(* CODESYS project mobject-types.library
   Company: mobject
   DefaultNamespace: mobject-types
   Version: 0.1.0
   Placeholder: mobject-types
   Author: mobject dev team
   Title: mobject-types

Project tree, tasks and I/O mapping:
  libraries: mobject-collections, 1.1.0 (mobject); mobject-deserialization, 0.1.0 (mobject); mobject-disposable, 1.0.0 (mobject); mobject-enumerable, 1.1.0 (mobject); mobject-serialization, 0.4.0 (mobject); Tc2_System, * (Beckhoff Automation GmbH); Tc2_Utilities, * (Beckhoff Automation GmbH)
  _Internal/
    Datatype/
      function block AliasDatatypeBase [ST]: AddBaseType, BaseType, Identifier, IecType, SerializeTypeWith, SerializeWith, TryDeserializeFrom, TryResolveAsAliasType
      function block DatatypeBase [ST]: Accept, Address, ClearReference, Clone, IecType, SerializeTypeWith, SerializeWith, Size, TryCopy, TryDeserializeFrom, TryMakeReferenceTo, TryResolveAsAliasType, TryResolveAsStructuredType
      function block StructuredDatatypeBase [ST]: AddMember, Accept, GetMemberEnumerator, Identifier, IecType, SerializeTypeWith, SerializeWith, TryCopy, TryDeserializeFrom, TryGetMemberByName, TryResolveAsStructuredType
    DatatypeVisitor/
      interface I_DatatypeVisitor: VisitDatatype
    MembersHost/
      interface I_HostMembers: TryGetMemberByName
      function block MembersHost [ST]: Accept, AddMember, GetMemberEnumerator, SerializeTypeWith, SerializeWith, TryDeserializeFrom, TryGetMemberByName
  Datatype/
    Alias/
      function block _HRESULT [ST]: FB_init, SetBaseTypeReference, Address, ClearReference, Clone, Identifier, MakeReferenceTo, Size, TryMakeReferenceTo, Value
      function block _FLOAT [ST]: FB_init, SetBaseTypeReference, Address, ClearReference, Clone, Identifier, MakeReferenceTo, Size, TryMakeReferenceTo, Value
    Primitive/
      function block _BOOL [ST]: FB_init, Address, ClearReference, Clone, IecType, MakeReferenceTo, SerializeWith, Size, TryDeserializeFrom, TryMakeReferenceTo, Value
      function block _BYTE [ST]: FB_init, Address, ClearReference, Clone, IecType, MakeReferenceTo, SerializeWith, Size, TryDeserializeFrom, TryMakeReferenceTo, Value
      function block _DINT [ST]: FB_init, Address, ClearReference, Clone, IecType, MakeReferenceTo, SerializeWith, Size, TryDeserializeFrom, TryMakeReferenceTo, Value
      function block _DT [ST]: FB_init, Address, ClearReference, Clone, IecType, MakeReferenceTo, SerializeWith, Size, TryDeserializeFrom, TryMakeReferenceTo, Value
      function block _DWORD [ST]: FB_init, Address, ClearReference, Clone, IecType, MakeReferenceTo, SerializeWith, Size, TryDeserializeFrom, TryMakeReferenceTo, Value
      function block _INT [ST]: FB_init, Address, ClearReference, Clone, IecType, MakeReferenceTo, SerializeWith, Size, TryDeserializeFrom, TryMakeReferenceTo, Value
      function block _LINT [ST]: FB_init, Address, ClearReference, Clone, IecType, MakeReferenceTo, SerializeWith, Size, TryDeserializeFrom, TryMakeReferenceTo, Value
      function block _LREAL [ST]: FB_init, Address, ClearReference, Clone, IecType, MakeReferenceTo, SerializeWith, Size, TryDeserializeFrom, TryMakeReferenceTo, Value
      function block _LWORD [ST]: FB_init, Address, ClearReference, Clone, IecType, MakeReferenceTo, SerializeWith, Size, TryDeserializeFrom, TryMakeReferenceTo, Value
      function block _REAL [ST]: FB_init, Address, ClearReference, Clone, IecType, MakeReferenceTo, SerializeWith, Size, TryDeserializeFrom, TryMakeReferenceTo, Value
      function block _SINT [ST]: FB_init, Address, ClearReference, Clone, IecType, MakeReferenceTo, SerializeWith, Size, TryDeserializeFrom, TryMakeReferenceTo, Value
      function block _TIME_OF_DAY [ST]: FB_init, Address, ClearReference, Clone, IecType, MakeReferenceTo, SerializeWith, Size, TryDeserializeFrom, TryMakeReferenceTo, Value
      function block _TOD [ST]: FB_init, Address, ClearReference, Clone, IecType, MakeReferenceTo, SerializeWith, Size, TryDeserializeFrom, TryMakeReferenceTo, Value
      function block _UDINT [ST]: FB_init, Address, ClearReference, Clone, IecType, MakeReferenceTo, SerializeWith, Size, TryDeserializeFrom, TryMakeReferenceTo, Value
      function block _UINT [ST]: FB_init, Address, ClearReference, Clone, IecType, MakeReferenceTo, SerializeWith, Size, TryDeserializeFrom, TryMakeReferenceTo, Value
      function block _ULINT [ST]: FB_init, Address, ClearReference, Clone, IecType, MakeReferenceTo, SerializeWith, Size, TryDeserializeFrom, TryMakeReferenceTo, Value
      function block _USINT [ST]: FB_init, Address, ClearReference, Clone, IecType, MakeReferenceTo, SerializeWith, Size, TryDeserializeFrom, TryMakeReferenceTo, Value
      function block _WORD [ST]: FB_init, Address, ClearReference, Clone, IecType, MakeReferenceTo, SerializeWith, Size, TryDeserializeFrom, TryMakeReferenceTo, Value
    Structs/
      function block _TIMESTRUCT [ST]: FB_init, SetMemberReference, Address, ClearReference, Clone, Identifier, MakeReferenceTo, Size, TryMakeReferenceTo, Value, wDay, wDayOfWeek, wHour, wMilliseconds, wMinute, wMonth, wSecond, wYear
  DatatypePacks/
    function block PlcBasicDatatypePack [ST]: RegisterWith
  Datatypes/
    Base/
    function block Datatypes [ST]: SerializeAliasTypeWith, SerializePrimitiveTypeWith, SerializeStructuresTypeWith, GetAliasByIdentifier, GetPrimitiveByIecType, GetStructureByIdentifier, RegisterDatatype, SerializeTypeWith
  Interfaces/
    interface I_AliasDatatype: BaseType, Identifier
    interface I_Datatype: Accept, Address, ClearReference, Clone, IecType, SerializeTypeWith, Size, TryDeserializeFrom, TryMakeReferenceTo, TryResolveAsAliasType, TryResolveAsStructuredType
    interface I_DatatypePack: RegisterWith
    interface I_Datatypes: GetAliasByIdentifier, GetPrimitiveByIecType, GetStructureByIdentifier, RegisterDatatype, SerializeTypeWith
    interface I_StructuredDatatype: Identifier, TryGetMemberByName
*)

// _Internal/Datatype/AliasDatatypeBase
FUNCTION_BLOCK ABSTRACT AliasDatatypeBase EXTENDS DatatypeBase IMPLEMENTS I_AliasDatatype
VAR
	_baseType : I_Datatype;
END_VAR

METHOD PROTECTED AddBaseType
VAR_INPUT
	BaseType : I_Datatype;
END_VAR
_baseType := BaseType;
END_METHOD

PROPERTY PUBLIC BaseType : I_Datatype
GET
BaseType := _baseType;
END_GET
END_PROPERTY

PROPERTY PUBLIC ABSTRACT Identifier : T_MAXSTRING
GET
END_GET
END_PROPERTY

PROPERTY PUBLIC IecType : T_MAXSTRING
GET
IecType := 'ALIAS';
END_GET
END_PROPERTY

METHOD PUBLIC SerializeTypeWith
VAR_INPUT
	Serializer : I_Serializer;
END_VAR
Serializer.StartObject();
Serializer.AddKeyString('name',Identifier);
Serializer.AddKeyString('type',IecType);
Serializer.AddKey('baseType');
_baseType.SerializeTypeWith(Serializer);
Serializer.EndObject();
END_METHOD

METHOD PUBLIC SerializeWith
VAR_INPUT
	Serializer : I_Serializer;
END_VAR
_baseType.SerializeWith(Serializer);
END_METHOD

METHOD TryDeserializeFrom : BOOL
VAR_INPUT
	Deserializer : I_Deserializer;
	Feedback : I_DeserializerFeedback;
END_VAR
TryDeserializeFrom := _baseType.TryDeserializeFrom(Deserializer, Feedback);
END_METHOD

METHOD PUBLIC TryResolveAsAliasType : BOOL
VAR_INPUT
	Destination : REFERENCE TO I_AliasDatatype;
END_VAR
Destination := THIS^;
TryResolveAsAliasType := TRUE;
END_METHOD

END_FUNCTION_BLOCK

// _Internal/Datatype/DatatypeBase
{attribute 'linkalways'} 
{attribute 'no_explicit_call' := 'This FB is a CLASS and must be accessed using methods or properties'}
{attribute 'enable_dynamic_creation'}
FUNCTION_BLOCK ABSTRACT DatatypeBase EXTENDS Disposable IMPLEMENTS I_Datatype
VAR
END_VAR

METHOD PUBLIC Accept
VAR_INPUT
	Visitor : I_DatatypeVisitor;
END_VAR
Visitor.VisitDatatype(this^);
END_METHOD

PROPERTY PUBLIC ABSTRACT Address : PVOID
GET
END_GET
END_PROPERTY

METHOD PUBLIC ABSTRACT ClearReference
VAR_INPUT
END_VAR
END_METHOD

METHOD PUBLIC ABSTRACT Clone : I_Datatype
END_METHOD

PROPERTY PUBLIC ABSTRACT IecType : T_MAXSTRING
GET
END_GET
END_PROPERTY

METHOD PUBLIC SerializeTypeWith
VAR_INPUT
	Serializer : I_Serializer;
END_VAR
Serializer.StartObject();
Serializer.AddKeyString('type',IecType);
Serializer.EndObject();
END_METHOD

METHOD PUBLIC ABSTRACT SerializeWith
VAR_INPUT
	Serializer : I_Serializer;
END_VAR
END_METHOD

PROPERTY PUBLIC ABSTRACT Size : UDINT
GET
END_GET
END_PROPERTY

METHOD PUBLIC TryCopy : BOOL
VAR_INPUT
	Source : I_Datatype;
END_VAR
IF Source.IecType <> IecType THEN
	RETURN;
END_IF

memcpy(Address, Source.Address, Size);
END_METHOD

METHOD PUBLIC ABSTRACT TryDeserializeFrom : BOOL
VAR_INPUT
	Deserializer : I_Deserializer;
	Feedback : I_DeserializerFeedback;
END_VAR
END_METHOD

METHOD PUBLIC ABSTRACT TryMakeReferenceTo : BOOL
VAR_INPUT
	Target : I_Datatype;
END_VAR
END_METHOD

METHOD PUBLIC TryResolveAsAliasType : BOOL
VAR_INPUT
	Destination : REFERENCE TO I_AliasDatatype;
END_VAR
TryResolveAsAliasType := FALSE;
RETURN;
END_METHOD

METHOD PUBLIC TryResolveAsStructuredType : BOOL
VAR_INPUT
	Destination : REFERENCE TO I_StructuredDatatype;
END_VAR
TryResolveAsStructuredType := FALSE;
RETURN;
END_METHOD

END_FUNCTION_BLOCK

// Interfaces/I_Datatype
INTERFACE I_Datatype extends I_Serializable, I_Deserializable, I_Disposable

METHOD PUBLIC Accept
VAR_INPUT
	Visitor : I_DatatypeVisitor;
END_VAR
END_METHOD

PROPERTY PUBLIC Address : PVOID
GET
END_GET
END_PROPERTY

METHOD PUBLIC ClearReference
VAR_INPUT
END_VAR
END_METHOD

METHOD Clone : I_Datatype
END_METHOD

PROPERTY PUBLIC IecType : T_MAXSTRING
GET
END_GET
END_PROPERTY

METHOD PUBLIC SerializeTypeWith
VAR_INPUT
	Serializer : I_Serializer;
END_VAR
END_METHOD

PROPERTY PUBLIC Size : UDINT
GET
END_GET
END_PROPERTY

METHOD PUBLIC ABSTRACT TryDeserializeFrom : BOOL
VAR_INPUT
	Deserializer : I_Deserializer;
	Feedback : I_DeserializerFeedback;
END_VAR
END_METHOD

METHOD TryMakeReferenceTo : BOOL
VAR_INPUT
	Target : I_Datatype;
END_VAR
END_METHOD

METHOD PUBLIC TryResolveAsAliasType : BOOL
VAR_INPUT
	Destination : REFERENCE TO I_AliasDatatype;
END_VAR
END_METHOD

METHOD PUBLIC TryResolveAsStructuredType : BOOL
VAR_INPUT
	Destination : REFERENCE TO I_StructuredDatatype;
END_VAR
END_METHOD

END_INTERFACE

// _Internal/DatatypeVisitor/I_DatatypeVisitor
INTERFACE I_DatatypeVisitor

METHOD VisitDatatype
VAR_INPUT
	VisitingDatatype : I_Datatype;
END_VAR
END_METHOD

END_INTERFACE

// Interfaces/I_AliasDatatype
INTERFACE I_AliasDatatype EXTENDS I_Datatype

PROPERTY PUBLIC BaseType : I_Datatype
GET
END_GET
END_PROPERTY

PROPERTY PUBLIC Identifier : T_MAXSTRING
GET
END_GET
END_PROPERTY

END_INTERFACE

// Interfaces/I_StructuredDatatype
INTERFACE I_StructuredDatatype EXTENDS I_Datatype

PROPERTY PUBLIC Identifier : T_MAXSTRING
GET
END_GET
END_PROPERTY

METHOD PUBLIC TryGetMemberByName : BOOL
VAR_INPUT
	Name : T_MAXSTRING;
	Destination : REFERENCE TO I_Datatype;
END_VAR
END_METHOD

END_INTERFACE

// _Internal/Datatype/StructuredDatatypeBase
{attribute 'linkalways'} 
{attribute 'no_explicit_call' := 'This FB is a CLASS and must be accessed using methods or properties'}
{attribute 'enable_dynamic_creation'}
FUNCTION_BLOCK ABSTRACT StructuredDatatypeBase EXTENDS DatatypeBase IMPLEMENTS I_StructuredDatatype
VAR
	membersHost : MembersHost;
END_VAR

METHOD PROTECTED AddMember
VAR_INPUT
	MemberName : T_MAXSTRING;
	Member : I_Datatype;
END_VAR
membersHost.AddMember(MemberName, Member);
END_METHOD

METHOD PUBLIC Accept
VAR_INPUT
	Visitor : I_DatatypeVisitor;
END_VAR
Visitor.VisitDatatype(THIS^);
membersHost.Accept(Visitor);
END_METHOD

METHOD PUBLIC GetMemberEnumerator : I_KeyValueForwardEnumerator
VAR_INPUT
END_VAR
GetMemberEnumerator := membersHost.GetMemberEnumerator();
END_METHOD

PROPERTY PUBLIC ABSTRACT Identifier : T_MAXSTRING
GET
END_GET
END_PROPERTY

PROPERTY PUBLIC IecType : T_MAXSTRING
GET
IecType := 'STRUCT';
END_GET
END_PROPERTY

METHOD PUBLIC SerializeTypeWith
VAR_INPUT
	Serializer : I_Serializer;
END_VAR
Serializer.StartObject();
Serializer.AddKeyString('name',Identifier);
Serializer.AddKeyString('type',IecType);	
membersHost.SerializeTypeWith(Serializer);
Serializer.EndObject();
END_METHOD

METHOD PUBLIC SerializeWith
VAR_INPUT
	Serializer : I_Serializer;
END_VAR
Serializer.StartObject();
membersHost.SerializeWith(Serializer);
Serializer.EndObject();
END_METHOD

METHOD PUBLIC TryCopy : BOOL
VAR_INPUT
	Source : I_Datatype;
END_VAR
VAR
	SourceAsStructure : I_StructuredDatatype;
END_VAR
IF NOT Source.TryResolveAsStructuredType(SourceAsStructure) THEN
	RETURN;
END_IF

IF SourceAsStructure.Identifier <> Identifier THEN
	RETURN;
END_IF

memcpy(Address, Source.Address, Size);
END_METHOD

METHOD TryDeserializeFrom : BOOL
VAR_INPUT
	Deserializer : I_Deserializer;
	Feedback : I_DeserializerFeedback;
END_VAR
TryDeserializeFrom := membersHost.TryDeserializeFrom(Deserializer, Feedback);
END_METHOD

METHOD PUBLIC TryGetMemberByName : BOOL
VAR_INPUT
	Name : T_MAXSTRING;
	Destination : REFERENCE TO I_Datatype;
END_VAR
VAR
	member : I_Datatype;
END_VAR
IF NOT membersHost.TryGetMemberByName(Name, member) THEN 
	RETURN;
END_IF

Destination := member;
TryGetMemberByName := TRUE;
END_METHOD

METHOD PUBLIC TryResolveAsStructuredType : BOOL
VAR_INPUT
	Destination : REFERENCE TO I_StructuredDatatype;
END_VAR
Destination := THIS^;
TryResolveAsStructuredType := TRUE;
END_METHOD

END_FUNCTION_BLOCK

// _Internal/MembersHost/MembersHost
{attribute 'linkalways'} 
{attribute 'no_explicit_call' := 'This FB is a CLASS and must be accessed using methods or properties'}
{attribute 'enable_dynamic_creation'}
FUNCTION_BLOCK MembersHost IMPLEMENTS I_Serializable
VAR
	members : Dictionary;
END_VAR

METHOD PUBLIC Accept
VAR_INPUT
	Visitor : I_DatatypeVisitor;
END_VAR
VAR
	enumerator : I_ForwardEnumerator;
	member : I_Datatype;
END_VAR
enumerator := members.GetEnumerator();

WHILE (enumerator.MoveNext()) DO
	
	IF enumerator.TryGet(member) THEN
		member.Accept(Visitor);
	END_IF

END_WHILE

enumerator.Dispose();
END_METHOD

METHOD PUBLIC AddMember
VAR_INPUT
	MemberName : T_MAXSTRING;
	Member : I_Datatype;
END_VAR
members.AddOrUpdate(MemberName, Member);
END_METHOD

METHOD PUBLIC GetMemberEnumerator : I_KeyValueForwardEnumerator
VAR_INPUT
END_VAR
GetMemberEnumerator := members.GetKeyValueEnumerator();
END_METHOD

METHOD PUBLIC SerializeTypeWith
VAR_INPUT
	Serializer : I_Serializer;
END_VAR
VAR
	enumerator : I_KeyValueForwardEnumerator;
	member : I_Datatype;
END_VAR
IF members.Count = 0 THEN
	RETURN;
END_IF

Serializer.AddKey('members');
Serializer.StartObject();

enumerator := members.GetKeyValueEnumerator();

WHILE enumerator.MoveNext() DO
	IF enumerator.TryGet(member) THEN
		Serializer.AddKey(enumerator.Key);
		member.SerializeTypeWith(Serializer);
	END_IF
END_WHILE

enumerator.Dispose();

Serializer.EndObject();
END_METHOD

METHOD PUBLIC SerializeWith
VAR_INPUT
	Serializer : I_Serializer;
END_VAR
VAR
	enumerator : I_KeyValueForwardEnumerator;
	member : I_Datatype;
END_VAR
enumerator := members.GetKeyValueEnumerator();

WHILE enumerator.MoveNext() DO
	IF enumerator.TryGet(member) THEN
		Serializer.AddKey(enumerator.Key);
		member.SerializeWith(Serializer);
	END_IF
END_WHILE

enumerator.Dispose();
END_METHOD

METHOD PUBLIC TryDeserializeFrom : BOOL
VAR_INPUT
	Deserializer : I_Deserializer;
	Feedback : I_DeserializerFeedback;
END_VAR
VAR
	membersEnumerator : I_DeserializerObjectForwardEnumerator;
	member : I_Datatype;
END_VAR
membersEnumerator := Deserializer.GetObjectEnumerator();

WHILE membersEnumerator.MoveNext() DO
	
	IF NOT TryGetMemberByName(membersEnumerator.Key, member) THEN
		CONTINUE;
	END_IF
	
	IF NOT member.TryDeserializeFrom(membersEnumerator.Current, Feedback) THEN
		RETURN;
	END_IF

END_WHILE

membersEnumerator.Dispose();
TryDeserializeFrom := TRUE;
END_METHOD

METHOD PUBLIC TryGetMemberByName : BOOL
VAR_INPUT
	Name : T_MAXSTRING;
	Destination : REFERENCE TO I_Datatype;
END_VAR
VAR
	member : I_Datatype;
END_VAR
IF NOT members.TryGetValue(Name, member) THEN
	RETURN;
END_IF

Destination := member;
TryGetMemberByName := TRUE;
END_METHOD

END_FUNCTION_BLOCK

// _Internal/MembersHost/I_HostMembers
INTERFACE I_HostMembers EXTENDS __SYSTEM.IQueryInterface

METHOD PUBLIC TryGetMemberByName : BOOL
VAR_INPUT
	Name : T_MAXSTRING;
	Destination : REFERENCE TO I_Datatype;
END_VAR
END_METHOD

END_INTERFACE

// Datatype/Alias/_HRESULT
{attribute 'linkalways'} 
{attribute 'no_explicit_call' := 'This FB is a CLASS and must be accessed using methods or properties'}
{attribute 'enable_dynamic_creation'}
FUNCTION_BLOCK _HRESULT EXTENDS AliasDatatypeBase
VAR
	localData : HRESULT;
	activeData : REFERENCE TO HRESULT REF= localData;
	aliasBaseType : _DINT(localData);
END_VAR

METHOD FB_init : BOOL
VAR_INPUT
	bInitRetains : BOOL; // if TRUE, the retain variables are initialized (warm start / cold start)
	bInCopyCode : BOOL;  // if TRUE, the instance afterwards gets moved into the copy code (online change)
	InitialValue : HRESULT;
END_VAR
localData := InitialValue;
SetBaseTypeReference();
AddBaseType(aliasBaseType);
END_METHOD

METHOD PROTECTED SetBaseTypeReference
VAR_INPUT
END_VAR
aliasBaseType.MakeReferenceTo(activeData);
END_METHOD

PROPERTY PUBLIC Address : PVOID
GET
Address := ADR(activeData);
END_GET
END_PROPERTY

METHOD PUBLIC ClearReference
VAR_INPUT
END_VAR
activeData REF= localData;
SetBaseTypeReference();
END_METHOD

METHOD PUBLIC Clone : I_Datatype
VAR
    pClone : POINTER TO _HRESULT;
END_VAR
pClone := __NEW(_HRESULT(InitialValue := Value));
Clone := pClone^;
END_METHOD

PROPERTY PUBLIC Identifier : T_MAXSTRING
GET
Identifier := 'HRESULT';
END_GET
END_PROPERTY

METHOD PUBLIC MakeReferenceTo
VAR_INPUT
	ReferenceTarget : REFERENCE TO HRESULT;
END_VAR
activeData REF= ReferenceTarget;
SetBaseTypeReference();
END_METHOD

PROPERTY PUBLIC Size : UDINT
GET
Size := SIZEOF(activeData);
END_GET
END_PROPERTY

METHOD TryMakeReferenceTo : BOOL
VAR_INPUT
	Target : I_Datatype;
END_VAR
VAR
	pTargetData : POINTER TO HRESULT;
END_VAR
IF NOT (Target.IecType = IecType) THEN
	RETURN;
END_IF

pTargetData := Target.Address;
activeData REF= pTargetData^;
SetBaseTypeReference();
TryMakeReferenceTo := TRUE;
END_METHOD

PROPERTY PUBLIC Value : HRESULT
GET
Value := activeData;
END_GET
SET
activeData := Value;
END_SET
END_PROPERTY

END_FUNCTION_BLOCK

// Datatype/Primitive/_DINT
{attribute 'linkalways'} 
{attribute 'no_explicit_call' := 'This FB is a CLASS and must be accessed using methods or properties'}
{attribute 'enable_dynamic_creation'}
FUNCTION_BLOCK _DINT EXTENDS DatatypeBase
VAR
	localData : DINT;
	activeData : REFERENCE TO DINT REF= localData;
END_VAR

METHOD FB_init : BOOL
VAR_INPUT
	bInitRetains : BOOL; // if TRUE, the retain variables are initialized (warm start / cold start)
	bInCopyCode : BOOL;  // if TRUE, the instance afterwards gets moved into the copy code (online change)
	InitialValue : DINT;
END_VAR
localData := InitialValue;
END_METHOD

PROPERTY PUBLIC Address : PVOID
GET
Address := ADR(activeData);
END_GET
END_PROPERTY

METHOD PUBLIC ClearReference
VAR_INPUT
END_VAR
activeData REF= localData;
END_METHOD

METHOD PUBLIC Clone : I_Datatype
VAR
    pClone : POINTER TO _DINT;
END_VAR
pClone := __NEW(_DINT(InitialValue := Value));
Clone := pClone^;
END_METHOD

PROPERTY PUBLIC IecType : T_MAXSTRING
GET
IecType := 'DINT';
END_GET
END_PROPERTY

METHOD PUBLIC MakeReferenceTo
VAR_INPUT
	ReferenceTarget : REFERENCE TO DINT;
END_VAR
activeData REF= ReferenceTarget;
END_METHOD

METHOD PUBLIC SerializeWith
VAR_INPUT
	Serializer : I_Serializer;
END_VAR
Serializer.AddDint(activeData);
END_METHOD

PROPERTY PUBLIC Size : UDINT
GET
Size := SIZEOF(activeData);
END_GET
END_PROPERTY

METHOD TryDeserializeFrom : BOOL
VAR_INPUT
	Deserializer : I_Deserializer;
	Feedback : I_DeserializerFeedback;
END_VAR
TryDeserializeFrom := Deserializer.TryGetDint(activeData, Feedback);
END_METHOD

METHOD TryMakeReferenceTo : BOOL
VAR_INPUT
	Target : I_Datatype;
END_VAR
VAR
	pTargetData : POINTER TO DINT;
END_VAR
IF NOT (Target.IecType = IecType) THEN
	RETURN;
END_IF

pTargetData := Target.Address;
activeData REF= pTargetData^;
TryMakeReferenceTo := TRUE;
END_METHOD

PROPERTY PUBLIC Value : DINT
GET
Value := activeData;
END_GET
SET
activeData := Value;
END_SET
END_PROPERTY

END_FUNCTION_BLOCK

// Datatype/Alias/_FLOAT
{attribute 'linkalways'} 
{attribute 'no_explicit_call' := 'This FB is a CLASS and must be accessed using methods or properties'}
{attribute 'enable_dynamic_creation'}
FUNCTION_BLOCK _FLOAT EXTENDS AliasDatatypeBase
VAR
	localData : FLOAT;
	activeData : REFERENCE TO FLOAT REF= localData;
	aliasBaseType : _LREAL(localData);
END_VAR

METHOD FB_init : BOOL
VAR_INPUT
	bInitRetains : BOOL; // if TRUE, the retain variables are initialized (warm start / cold start)
	bInCopyCode : BOOL;  // if TRUE, the instance afterwards gets moved into the copy code (online change)
	InitialValue : FLOAT;
END_VAR
localData := InitialValue;
SetBaseTypeReference();
AddBaseType(aliasBaseType);
END_METHOD

METHOD PROTECTED SetBaseTypeReference
VAR_INPUT
END_VAR
aliasBaseType.MakeReferenceTo(activeData);
END_METHOD

PROPERTY PUBLIC Address : PVOID
GET
Address := ADR(activeData);
END_GET
END_PROPERTY

METHOD PUBLIC ClearReference
VAR_INPUT
END_VAR
activeData REF= localData;
SetBaseTypeReference();
END_METHOD

METHOD PUBLIC Clone : I_Datatype
VAR
    pClone : POINTER TO _FLOAT;
END_VAR
pClone := __NEW(_FLOAT(InitialValue := Value));
Clone := pClone^;
END_METHOD

PROPERTY PUBLIC Identifier : T_MAXSTRING
GET
Identifier := 'FLOAT';
END_GET
END_PROPERTY

METHOD PUBLIC MakeReferenceTo
VAR_INPUT
	ReferenceTarget : REFERENCE TO FLOAT;
END_VAR
activeData REF= ReferenceTarget;
SetBaseTypeReference();
END_METHOD

PROPERTY PUBLIC Size : UDINT
GET
Size := SIZEOF(activeData);
END_GET
END_PROPERTY

METHOD TryMakeReferenceTo : BOOL
VAR_INPUT
	Target : I_Datatype;
END_VAR
VAR
	pTargetData : POINTER TO FLOAT;
END_VAR
IF NOT (Target.IecType = IecType) THEN
	RETURN;
END_IF

pTargetData := Target.Address;
activeData REF= pTargetData^;
SetBaseTypeReference();
TryMakeReferenceTo := TRUE;
END_METHOD

PROPERTY PUBLIC Value : FLOAT
GET
Value := activeData;
END_GET
SET
activeData := Value;
END_SET
END_PROPERTY

END_FUNCTION_BLOCK

// Datatype/Primitive/_LREAL
{attribute 'linkalways'} 
{attribute 'no_explicit_call' := 'This FB is a CLASS and must be accessed using methods or properties'}
{attribute 'enable_dynamic_creation'}
FUNCTION_BLOCK _LREAL EXTENDS DatatypeBase
VAR
	localData : LREAL;
	activeData : REFERENCE TO LREAL REF= localData;
END_VAR

METHOD FB_init : BOOL
VAR_INPUT
	bInitRetains : BOOL; // if TRUE, the retain variables are initialized (warm start / cold start)
	bInCopyCode : BOOL;  // if TRUE, the instance afterwards gets moved into the copy code (online change)
	InitialValue : LREAL;
END_VAR
localData := InitialValue;
END_METHOD

PROPERTY PUBLIC Address : PVOID
GET
Address := ADR(activeData);
END_GET
END_PROPERTY

METHOD PUBLIC ClearReference
VAR_INPUT
END_VAR
activeData REF= localData;
END_METHOD

METHOD PUBLIC Clone : I_Datatype
VAR
    pClone : POINTER TO _LREAL;
END_VAR
pClone := __NEW(_LREAL(InitialValue := Value));
Clone := pClone^;
END_METHOD

PROPERTY PUBLIC IecType : T_MAXSTRING
GET
IecType := 'LREAL';
END_GET
END_PROPERTY

METHOD PUBLIC MakeReferenceTo
VAR_INPUT
	ReferenceTarget : REFERENCE TO LREAL;
END_VAR
activeData REF= ReferenceTarget;
END_METHOD

METHOD PUBLIC SerializeWith
VAR_INPUT
	Serializer : I_Serializer;
END_VAR
Serializer.AddLreal(activeData);
END_METHOD

PROPERTY PUBLIC Size : UDINT
GET
Size := SIZEOF(activeData);
END_GET
END_PROPERTY

METHOD TryDeserializeFrom : BOOL
VAR_INPUT
	Deserializer : I_Deserializer;
	Feedback : I_DeserializerFeedback;
END_VAR
TryDeserializeFrom := Deserializer.TryGetLreal(activeData, Feedback);
END_METHOD

METHOD TryMakeReferenceTo : BOOL
VAR_INPUT
	Target : I_Datatype;
END_VAR
VAR
	pTargetData : POINTER TO LREAL;
END_VAR
IF NOT (Target.IecType = IecType) THEN
	RETURN;
END_IF

pTargetData := Target.Address;
activeData REF= pTargetData^;
TryMakeReferenceTo := TRUE;
END_METHOD

PROPERTY PUBLIC Value : LREAL
GET
Value := activeData;
END_GET
SET
activeData := Value;
END_SET
END_PROPERTY

END_FUNCTION_BLOCK

// Datatype/Primitive/_BOOL
{attribute 'linkalways'} 
{attribute 'no_explicit_call' := 'This FB is a CLASS and must be accessed using methods or properties'}
{attribute 'enable_dynamic_creation'}
FUNCTION_BLOCK _BOOL EXTENDS DatatypeBase
VAR
	localData : BOOL;
	activeData : REFERENCE TO BOOL REF= localData;
END_VAR

METHOD FB_init : BOOL
VAR_INPUT
	bInitRetains : BOOL; // if TRUE, the retain variables are initialized (warm start / cold start)
	bInCopyCode : BOOL;  // if TRUE, the instance afterwards gets moved into the copy code (online change)
	InitialValue : BOOL;
END_VAR
localData := InitialValue;
END_METHOD

PROPERTY PUBLIC Address : PVOID
GET
Address := ADR(activeData);
END_GET
END_PROPERTY

METHOD PUBLIC ClearReference
VAR_INPUT
END_VAR
activeData REF= localData;
END_METHOD

METHOD PUBLIC Clone : I_Datatype
VAR
    pClone : POINTER TO _BOOL;
END_VAR
pClone := __NEW(_BOOL(InitialValue := Value));
Clone := pClone^;
END_METHOD

PROPERTY PUBLIC IecType : T_MAXSTRING
GET
IecType := 'BOOL';
END_GET
END_PROPERTY

METHOD PUBLIC MakeReferenceTo
VAR_INPUT
	ReferenceTarget : REFERENCE TO BOOL;
END_VAR
activeData REF= ReferenceTarget;
END_METHOD

METHOD PUBLIC SerializeWith
VAR_INPUT
	Serializer : I_Serializer;
END_VAR
Serializer.AddBool(activeData);
END_METHOD

PROPERTY PUBLIC Size : UDINT
GET
Size := SIZEOF(activeData);
END_GET
END_PROPERTY

METHOD TryDeserializeFrom : BOOL
VAR_INPUT
	Deserializer : I_Deserializer;
	Feedback : I_DeserializerFeedback;
END_VAR
TryDeserializeFrom := Deserializer.TryGetBool(activeData, Feedback);
END_METHOD

METHOD TryMakeReferenceTo : BOOL
VAR_INPUT
	Target : I_Datatype;
END_VAR
VAR
	pTargetData : POINTER TO BOOL;
END_VAR
IF NOT (Target.IecType = IecType) THEN
	RETURN;
END_IF

pTargetData := Target.Address;
activeData REF= pTargetData^;
TryMakeReferenceTo := TRUE;
END_METHOD

PROPERTY PUBLIC Value : BOOL
GET
Value := activeData;
END_GET
SET
activeData := Value;
END_SET
END_PROPERTY

END_FUNCTION_BLOCK

// Datatype/Primitive/_BYTE
{attribute 'linkalways'} 
{attribute 'no_explicit_call' := 'This FB is a CLASS and must be accessed using methods or properties'}
{attribute 'enable_dynamic_creation'}
FUNCTION_BLOCK _BYTE EXTENDS DatatypeBase
VAR
	localData : BYTE;
	activeData : REFERENCE TO BYTE REF= localData;
END_VAR

METHOD FB_init : BOOL
VAR_INPUT
	bInitRetains : BOOL; // if TRUE, the retain variables are initialized (warm start / cold start)
	bInCopyCode : BOOL;  // if TRUE, the instance afterwards gets moved into the copy code (online change)
	InitialValue : BYTE;
END_VAR
localData := InitialValue;
END_METHOD

PROPERTY PUBLIC Address : PVOID
GET
Address := ADR(activeData);
END_GET
END_PROPERTY

METHOD PUBLIC ClearReference
VAR_INPUT
END_VAR
activeData REF= localData;
END_METHOD

METHOD PUBLIC Clone : I_Datatype
VAR
    pClone : POINTER TO _BYTE;
END_VAR
pClone := __NEW(_BYTE(InitialValue := Value));
Clone := pClone^;
END_METHOD

PROPERTY PUBLIC IecType : T_MAXSTRING
GET
IecType := 'BYTE';
END_GET
END_PROPERTY

METHOD PUBLIC MakeReferenceTo
VAR_INPUT
	ReferenceTarget : REFERENCE TO BYTE;
END_VAR
activeData REF= ReferenceTarget;
END_METHOD

METHOD PUBLIC SerializeWith
VAR_INPUT
	Serializer : I_Serializer;
END_VAR
Serializer.AddByte(activeData);
END_METHOD

PROPERTY PUBLIC Size : UDINT
GET
Size := SIZEOF(activeData);
END_GET
END_PROPERTY

METHOD TryDeserializeFrom : BOOL
VAR_INPUT
	Deserializer : I_Deserializer;
	Feedback : I_DeserializerFeedback;
END_VAR
TryDeserializeFrom := Deserializer.TryGetByte(activeData, Feedback);
END_METHOD

METHOD TryMakeReferenceTo : BOOL
VAR_INPUT
	Target : I_Datatype;
END_VAR
VAR
	pTargetData : POINTER TO BYTE;
END_VAR
IF NOT (Target.IecType = IecType) THEN
	RETURN;
END_IF

pTargetData := Target.Address;
activeData REF= pTargetData^;
TryMakeReferenceTo := TRUE;
END_METHOD

PROPERTY PUBLIC Value : BYTE
GET
Value := activeData;
END_GET
SET
activeData := Value;
END_SET
END_PROPERTY

END_FUNCTION_BLOCK

// Datatype/Primitive/_DT
{attribute 'linkalways'} 
{attribute 'no_explicit_call' := 'This FB is a CLASS and must be accessed using methods or properties'}
{attribute 'enable_dynamic_creation'}
FUNCTION_BLOCK _DT EXTENDS DatatypeBase
VAR
	localData : DT;
	activeData : REFERENCE TO DT REF= localData;
END_VAR

METHOD FB_init : BOOL
VAR_INPUT
	bInitRetains : BOOL; // if TRUE, the retain variables are initialized (warm start / cold start)
	bInCopyCode : BOOL;  // if TRUE, the instance afterwards gets moved WORDo the copy code (online change)
	InitialValue : DT;
END_VAR
localData := InitialValue;
END_METHOD

PROPERTY PUBLIC Address : PVOID
GET
Address := ADR(activeData);
END_GET
END_PROPERTY

METHOD PUBLIC ClearReference
VAR_INPUT
END_VAR
activeData REF= localData;
END_METHOD

METHOD PUBLIC Clone : I_Datatype
VAR
    pClone : POINTER TO _DT;
END_VAR
pClone := __NEW(_DT(InitialValue := Value));
Clone := pClone^;
END_METHOD

PROPERTY PUBLIC IecType : T_MAXSTRING
GET
IecType := 'DT';
END_GET
END_PROPERTY

METHOD PUBLIC MakeReferenceTo
VAR_INPUT
	ReferenceTarget : REFERENCE TO DT;
END_VAR
activeData REF= ReferenceTarget;
END_METHOD

METHOD PUBLIC SerializeWith
VAR_INPUT
	Serializer : I_Serializer;
END_VAR
Serializer.AddDateTime(activeData);
END_METHOD

PROPERTY PUBLIC Size : UDINT
GET
Size := SIZEOF(activeData);
END_GET
END_PROPERTY

METHOD TryDeserializeFrom : BOOL
VAR_INPUT
	Deserializer : I_Deserializer;
	Feedback : I_DeserializerFeedback;
END_VAR
TryDeserializeFrom := Deserializer.TryGetDateTime(activeData, Feedback);
END_METHOD

METHOD TryMakeReferenceTo : BOOL
VAR_INPUT
	Target : I_Datatype;
END_VAR
VAR
	pTargetData : POINTER TO DT;
END_VAR
IF NOT (Target.IecType = IecType) THEN
	RETURN;
END_IF

pTargetData := Target.Address;
activeData REF= pTargetData^;
TryMakeReferenceTo := TRUE;
END_METHOD

PROPERTY PUBLIC Value : DT
GET
Value := activeData;
END_GET
SET
activeData := Value;
END_SET
END_PROPERTY

END_FUNCTION_BLOCK

// Datatype/Primitive/_DWORD
{attribute 'linkalways'} 
{attribute 'no_explicit_call' := 'This FB is a CLASS and must be accessed using methods or properties'}
{attribute 'enable_dynamic_creation'}
FUNCTION_BLOCK _DWORD EXTENDS DatatypeBase
VAR
	localData : DWORD;
	activeData : REFERENCE TO DWORD REF= localData;
END_VAR

METHOD FB_init : BOOL
VAR_INPUT
	bInitRetains : BOOL; // if TRUE, the retain variables are initialized (warm start / cold start)
	bInCopyCode : BOOL;  // if TRUE, the instance afterwards gets moved WORDo the copy code (online change)
	InitialValue : DWORD;
END_VAR
localData := InitialValue;
END_METHOD

PROPERTY PUBLIC Address : PVOID
GET
Address := ADR(activeData);
END_GET
END_PROPERTY

METHOD PUBLIC ClearReference
VAR_INPUT
END_VAR
activeData REF= localData;
END_METHOD

METHOD PUBLIC Clone : I_Datatype
VAR
    pClone : POINTER TO _DWORD;
END_VAR
pClone := __NEW(_DWORD(InitialValue := Value));
Clone := pClone^;
END_METHOD

PROPERTY PUBLIC IecType : T_MAXSTRING
GET
IecType := 'DWORD';
END_GET
END_PROPERTY

METHOD PUBLIC MakeReferenceTo
VAR_INPUT
	ReferenceTarget : REFERENCE TO DWORD;
END_VAR
activeData REF= ReferenceTarget;
END_METHOD

METHOD PUBLIC SerializeWith
VAR_INPUT
	Serializer : I_Serializer;
END_VAR
Serializer.AddDword(activeData);
END_METHOD

PROPERTY PUBLIC Size : UDINT
GET
Size := SIZEOF(activeData);
END_GET
END_PROPERTY

METHOD TryDeserializeFrom : BOOL
VAR_INPUT
	Deserializer : I_Deserializer;
	Feedback : I_DeserializerFeedback;
END_VAR
TryDeserializeFrom := Deserializer.TryGetDword(activeData, Feedback);
END_METHOD

METHOD TryMakeReferenceTo : BOOL
VAR_INPUT
	Target : I_Datatype;
END_VAR
VAR
	pTargetData : POINTER TO DWORD;
END_VAR
IF NOT (Target.IecType = IecType) THEN
	RETURN;
END_IF

pTargetData := Target.Address;
activeData REF= pTargetData^;
TryMakeReferenceTo := TRUE;
END_METHOD

PROPERTY PUBLIC Value : DWORD
GET
Value := activeData;
END_GET
SET
activeData := Value;
END_SET
END_PROPERTY

END_FUNCTION_BLOCK

// Datatype/Primitive/_INT
{attribute 'linkalways'} 
{attribute 'no_explicit_call' := 'This FB is a CLASS and must be accessed using methods or properties'}
{attribute 'enable_dynamic_creation'}
FUNCTION_BLOCK _INT EXTENDS DatatypeBase
VAR
	localData : INT;
	activeData : REFERENCE TO INT REF= localData;
END_VAR

METHOD FB_init : BOOL
VAR_INPUT
	bInitRetains : BOOL; // if TRUE, the retain variables are initialized (warm start / cold start)
	bInCopyCode : BOOL;  // if TRUE, the instance afterwards gets moved into the copy code (online change)
	InitialValue : INT;
END_VAR
localData := InitialValue;
END_METHOD

PROPERTY PUBLIC Address : PVOID
GET
Address := ADR(activeData);
END_GET
END_PROPERTY

METHOD PUBLIC ClearReference
VAR_INPUT
END_VAR
activeData REF= localData;
END_METHOD

METHOD PUBLIC Clone : I_Datatype
VAR
    pClone : POINTER TO _INT;
END_VAR
pClone := __NEW(_INT(InitialValue := Value));
Clone := pClone^;
END_METHOD

PROPERTY PUBLIC IecType : T_MAXSTRING
GET
IecType := 'INT';
END_GET
END_PROPERTY

METHOD PUBLIC MakeReferenceTo
VAR_INPUT
	ReferenceTarget : REFERENCE TO INT;
END_VAR
activeData REF= ReferenceTarget;
END_METHOD

METHOD PUBLIC SerializeWith
VAR_INPUT
	Serializer : I_Serializer;
END_VAR
Serializer.AddInt(activeData);
END_METHOD

PROPERTY PUBLIC Size : UDINT
GET
Size := SIZEOF(activeData);
END_GET
END_PROPERTY

METHOD TryDeserializeFrom : BOOL
VAR_INPUT
	Deserializer : I_Deserializer;
	Feedback : I_DeserializerFeedback;
END_VAR
TryDeserializeFrom := Deserializer.TryGetInt(activeData, Feedback);
END_METHOD

METHOD TryMakeReferenceTo : BOOL
VAR_INPUT
	Target : I_Datatype;
END_VAR
VAR
	pTargetData : POINTER TO INT;
END_VAR
IF NOT (Target.IecType = IecType) THEN
	RETURN;
END_IF

pTargetData := Target.Address;
activeData REF= pTargetData^;
TryMakeReferenceTo := TRUE;
END_METHOD

PROPERTY PUBLIC Value : INT
GET
Value := activeData;
END_GET
SET
activeData := Value;
END_SET
END_PROPERTY

END_FUNCTION_BLOCK

// Datatype/Primitive/_LINT
{attribute 'linkalways'} 
{attribute 'no_explicit_call' := 'This FB is a CLASS and must be accessed using methods or properties'}
{attribute 'enable_dynamic_creation'}
FUNCTION_BLOCK _LINT EXTENDS DatatypeBase
VAR
	localData : LINT;
	activeData : REFERENCE TO LINT REF= localData;
END_VAR

METHOD FB_init : BOOL
VAR_INPUT
	bInitRetains : BOOL; // if TRUE, the retain variables are initialized (warm start / cold start)
	bInCopyCode : BOOL;  // if TRUE, the instance afterwards gets moved into the copy code (online change)
	InitialValue : LINT;
END_VAR
localData := InitialValue;
END_METHOD

PROPERTY PUBLIC Address : PVOID
GET
Address := ADR(activeData);
END_GET
END_PROPERTY

METHOD PUBLIC ClearReference
VAR_INPUT
END_VAR
activeData REF= localData;
END_METHOD

METHOD PUBLIC Clone : I_Datatype
VAR
    pClone : POINTER TO _LINT;
END_VAR
pClone := __NEW(_LINT(InitialValue := Value));
Clone := pClone^;
END_METHOD

PROPERTY PUBLIC IecType : T_MAXSTRING
GET
IecType := 'LINT';
END_GET
END_PROPERTY

METHOD PUBLIC MakeReferenceTo
VAR_INPUT
	ReferenceTarget : REFERENCE TO LINT;
END_VAR
activeData REF= ReferenceTarget;
END_METHOD

METHOD PUBLIC SerializeWith
VAR_INPUT
	Serializer : I_Serializer;
END_VAR
Serializer.AddLint(activeData);
END_METHOD

PROPERTY PUBLIC Size : UDINT
GET
Size := SIZEOF(activeData);
END_GET
END_PROPERTY

METHOD TryDeserializeFrom : BOOL
VAR_INPUT
	Deserializer : I_Deserializer;
	Feedback : I_DeserializerFeedback;
END_VAR
TryDeserializeFrom := Deserializer.TryGetLint(activeData, Feedback);
END_METHOD

METHOD TryMakeReferenceTo : BOOL
VAR_INPUT
	Target : I_Datatype;
END_VAR
VAR
	pTargetData : POINTER TO LINT;
END_VAR
IF NOT (Target.IecType = IecType) THEN
	RETURN;
END_IF

pTargetData := Target.Address;
activeData REF= pTargetData^;
TryMakeReferenceTo := TRUE;
END_METHOD

PROPERTY PUBLIC Value : LINT
GET
Value := activeData;
END_GET
SET
activeData := Value;
END_SET
END_PROPERTY

END_FUNCTION_BLOCK

// Datatype/Primitive/_LWORD
{attribute 'linkalways'} 
{attribute 'no_explicit_call' := 'This FB is a CLASS and must be accessed using methods or properties'}
{attribute 'enable_dynamic_creation'}
FUNCTION_BLOCK _LWORD EXTENDS DatatypeBase
VAR
	localData : LWORD;
	activeData : REFERENCE TO LWORD REF= localData;
END_VAR

METHOD FB_init : BOOL
VAR_INPUT
	bInitRetains : BOOL; // if TRUE, the retain variables are initialized (warm start / cold start)
	bInCopyCode : BOOL;  // if TRUE, the instance afterwards gets moved WORDo the copy code (online change)
	InitialValue : LWORD;
END_VAR
localData := InitialValue;
END_METHOD

PROPERTY PUBLIC Address : PVOID
GET
Address := ADR(activeData);
END_GET
END_PROPERTY

METHOD PUBLIC ClearReference
VAR_INPUT
END_VAR
activeData REF= localData;
END_METHOD

METHOD PUBLIC Clone : I_Datatype
VAR
    pClone : POINTER TO _LWORD;
END_VAR
pClone := __NEW(_LWORD(InitialValue := Value));
Clone := pClone^;
END_METHOD

PROPERTY PUBLIC IecType : T_MAXSTRING
GET
IecType := 'LWORD';
END_GET
END_PROPERTY

METHOD PUBLIC MakeReferenceTo
VAR_INPUT
	ReferenceTarget : REFERENCE TO LWORD;
END_VAR
activeData REF= ReferenceTarget;
END_METHOD

METHOD PUBLIC SerializeWith
VAR_INPUT
	Serializer : I_Serializer;
END_VAR
Serializer.AddLword(activeData);
END_METHOD

PROPERTY PUBLIC Size : UDINT
GET
Size := SIZEOF(activeData);
END_GET
END_PROPERTY

METHOD TryDeserializeFrom : BOOL
VAR_INPUT
	Deserializer : I_Deserializer;
	Feedback : I_DeserializerFeedback;
END_VAR
TryDeserializeFrom := Deserializer.TryGetLword(activeData, Feedback);
END_METHOD

METHOD TryMakeReferenceTo : BOOL
VAR_INPUT
	Target : I_Datatype;
END_VAR
VAR
	pTargetData : POINTER TO LWORD;
END_VAR
IF NOT (Target.IecType = IecType) THEN
	RETURN;
END_IF

pTargetData := Target.Address;
activeData REF= pTargetData^;
TryMakeReferenceTo := TRUE;
END_METHOD

PROPERTY PUBLIC Value : LWORD
GET
Value := activeData;
END_GET
SET
activeData := Value;
END_SET
END_PROPERTY

END_FUNCTION_BLOCK

// Datatype/Primitive/_REAL
{attribute 'linkalways'} 
{attribute 'no_explicit_call' := 'This FB is a CLASS and must be accessed using methods or properties'}
{attribute 'enable_dynamic_creation'}
FUNCTION_BLOCK _REAL EXTENDS DatatypeBase
VAR
	localData : REAL;
	activeData : REFERENCE TO REAL REF= localData;
END_VAR

METHOD FB_init : BOOL
VAR_INPUT
	bInitRetains : BOOL; // if TRUE, the retain variables are initialized (warm start / cold start)
	bInCopyCode : BOOL;  // if TRUE, the instance afterwards gets moved into the copy code (online change)
	InitialValue : REAL;
END_VAR
localData := InitialValue;
END_METHOD

PROPERTY PUBLIC Address : PVOID
GET
Address := ADR(activeData);
END_GET
END_PROPERTY

METHOD PUBLIC ClearReference
VAR_INPUT
END_VAR
activeData REF= localData;
END_METHOD

METHOD PUBLIC Clone : I_Datatype
VAR
    pClone : POINTER TO _REAL;
END_VAR
pClone := __NEW(_REAL(InitialValue := Value));
Clone := pClone^;
END_METHOD

PROPERTY PUBLIC IecType : T_MAXSTRING
GET
IecType := 'REAL';
END_GET
END_PROPERTY

METHOD PUBLIC MakeReferenceTo
VAR_INPUT
	ReferenceTarget : REFERENCE TO REAL;
END_VAR
activeData REF= ReferenceTarget;
END_METHOD

METHOD PUBLIC SerializeWith
VAR_INPUT
	Serializer : I_Serializer;
END_VAR
Serializer.AddReal(activeData);
END_METHOD

PROPERTY PUBLIC Size : UDINT
GET
Size := SIZEOF(activeData);
END_GET
END_PROPERTY

METHOD TryDeserializeFrom : BOOL
VAR_INPUT
	Deserializer : I_Deserializer;
	Feedback : I_DeserializerFeedback;
END_VAR
TryDeserializeFrom := Deserializer.TryGetReal(activeData, Feedback);
END_METHOD

METHOD TryMakeReferenceTo : BOOL
VAR_INPUT
	Target : I_Datatype;
END_VAR
VAR
	pTargetData : POINTER TO REAL;
END_VAR
IF NOT (Target.IecType = IecType) THEN
	RETURN;
END_IF

pTargetData := Target.Address;
activeData REF= pTargetData^;
TryMakeReferenceTo := TRUE;
END_METHOD

PROPERTY PUBLIC Value : REAL
GET
Value := activeData;
END_GET
SET
activeData := Value;
END_SET
END_PROPERTY

END_FUNCTION_BLOCK

// Datatype/Primitive/_SINT
{attribute 'linkalways'} 
{attribute 'no_explicit_call' := 'This FB is a CLASS and must be accessed using methods or properties'}
{attribute 'enable_dynamic_creation'}
FUNCTION_BLOCK _SINT EXTENDS DatatypeBase
VAR
	localData : SINT;
	activeData : REFERENCE TO SINT REF= localData;
END_VAR

METHOD FB_init : BOOL
VAR_INPUT
	bInitRetains : BOOL; // if TRUE, the retain variables are initialized (warm start / cold start)
	bInCopyCode : BOOL;  // if TRUE, the instance afterwards gets moved into the copy code (online change)
	InitialValue : SINT;
END_VAR
localData := InitialValue;
END_METHOD

PROPERTY PUBLIC Address : PVOID
GET
Address := ADR(activeData);
END_GET
END_PROPERTY

METHOD PUBLIC ClearReference
VAR_INPUT
END_VAR
activeData REF= localData;
END_METHOD

METHOD PUBLIC Clone : I_Datatype
VAR
    pClone : POINTER TO _SINT;
END_VAR
pClone := __NEW(_SINT(InitialValue := Value));
Clone := pClone^;
END_METHOD

PROPERTY PUBLIC IecType : T_MAXSTRING
GET
IecType := 'SINT';
END_GET
END_PROPERTY

METHOD PUBLIC MakeReferenceTo
VAR_INPUT
	ReferenceTarget : REFERENCE TO SINT;
END_VAR
activeData REF= ReferenceTarget;
END_METHOD

METHOD PUBLIC SerializeWith
VAR_INPUT
	Serializer : I_Serializer;
END_VAR
Serializer.AddSint(activeData);
END_METHOD

PROPERTY PUBLIC Size : UDINT
GET
Size := SIZEOF(activeData);
END_GET
END_PROPERTY

METHOD TryDeserializeFrom : BOOL
VAR_INPUT
	Deserializer : I_Deserializer;
	Feedback : I_DeserializerFeedback;
END_VAR
TryDeserializeFrom := Deserializer.TryGetSint(activeData, Feedback);
END_METHOD

METHOD TryMakeReferenceTo : BOOL
VAR_INPUT
	Target : I_Datatype;
END_VAR
VAR
	pTargetData : POINTER TO SINT;
END_VAR
IF NOT (Target.IecType = IecType) THEN
	RETURN;
END_IF

pTargetData := Target.Address;
activeData REF= pTargetData^;
TryMakeReferenceTo := TRUE;
END_METHOD

PROPERTY PUBLIC Value : SINT
GET
Value := activeData;
END_GET
SET
activeData := Value;
END_SET
END_PROPERTY

END_FUNCTION_BLOCK

// Datatype/Primitive/_TIME_OF_DAY
{attribute 'linkalways'} 
{attribute 'no_explicit_call' := 'This FB is a CLASS and must be accessed using methods or properties'}
{attribute 'enable_dynamic_creation'}
FUNCTION_BLOCK _TIME_OF_DAY EXTENDS DatatypeBase
VAR
	localData : TIME_OF_DAY;
	activeData : REFERENCE TO TIME_OF_DAY REF= localData;
END_VAR

METHOD FB_init : BOOL
VAR_INPUT
	bInitRetains : BOOL; // if TRUE, the retain variables are initialized (warm start / cold start)
	bInCopyCode : BOOL;  // if TRUE, the instance afterwards gets moved WORDo the copy code (online change)
	InitialValue : TIME_OF_DAY;
END_VAR
localData := InitialValue;
END_METHOD

PROPERTY PUBLIC Address : PVOID
GET
Address := ADR(activeData);
END_GET
END_PROPERTY

METHOD PUBLIC ClearReference
VAR_INPUT
END_VAR
activeData REF= localData;
END_METHOD

METHOD PUBLIC Clone : I_Datatype
VAR
    pClone : POINTER TO _TIME_OF_DAY;
END_VAR
pClone := __NEW(_TIME_OF_DAY(InitialValue := Value));
Clone := pClone^;
END_METHOD

PROPERTY PUBLIC IecType : T_MAXSTRING
GET
IecType := 'TIME_OF_DAY';
END_GET
END_PROPERTY

METHOD PUBLIC MakeReferenceTo
VAR_INPUT
	ReferenceTarget : REFERENCE TO TIME_OF_DAY;
END_VAR
activeData REF= ReferenceTarget;
END_METHOD

METHOD PUBLIC SerializeWith
VAR_INPUT
	Serializer : I_Serializer;
END_VAR
Serializer.AddTod(activeData);
END_METHOD

PROPERTY PUBLIC Size : UDINT
GET
Size := SIZEOF(activeData);
END_GET
END_PROPERTY

METHOD TryDeserializeFrom : BOOL
VAR_INPUT
	Deserializer : I_Deserializer;
	Feedback : I_DeserializerFeedback;
END_VAR
TryDeserializeFrom := Deserializer.TryGetTod(activeData, Feedback);
END_METHOD

METHOD TryMakeReferenceTo : BOOL
VAR_INPUT
	Target : I_Datatype;
END_VAR
VAR
	pTargetData : POINTER TO TIME_OF_DAY;
END_VAR
IF NOT (Target.IecType = IecType) THEN
	RETURN;
END_IF

pTargetData := Target.Address;
activeData REF= pTargetData^;
TryMakeReferenceTo := TRUE;
END_METHOD

PROPERTY PUBLIC Value : TIME_OF_DAY
GET
Value := activeData;
END_GET
SET
activeData := Value;
END_SET
END_PROPERTY

END_FUNCTION_BLOCK

// Datatype/Primitive/_TOD
{attribute 'linkalways'} 
{attribute 'no_explicit_call' := 'This FB is a CLASS and must be accessed using methods or properties'}
{attribute 'enable_dynamic_creation'}
FUNCTION_BLOCK _TOD EXTENDS DatatypeBase
VAR
	localData : TOD;
	activeData : REFERENCE TO TOD REF= localData;
END_VAR

METHOD FB_init : BOOL
VAR_INPUT
	bInitRetains : BOOL; // if TRUE, the retain variables are initialized (warm start / cold start)
	bInCopyCode : BOOL;  // if TRUE, the instance afterwards gets moved WORDo the copy code (online change)
	InitialValue : TOD;
END_VAR
localData := InitialValue;
END_METHOD

PROPERTY PUBLIC Address : PVOID
GET
Address := ADR(activeData);
END_GET
END_PROPERTY

METHOD PUBLIC ClearReference
VAR_INPUT
END_VAR
activeData REF= localData;
END_METHOD

METHOD PUBLIC Clone : I_Datatype
VAR
    pClone : POINTER TO _TOD;
END_VAR
pClone := __NEW(_TOD(InitialValue := Value));
Clone := pClone^;
END_METHOD

PROPERTY PUBLIC IecType : T_MAXSTRING
GET
IecType := 'TOD';
END_GET
END_PROPERTY

METHOD PUBLIC MakeReferenceTo
VAR_INPUT
	ReferenceTarget : REFERENCE TO TOD;
END_VAR
activeData REF= ReferenceTarget;
END_METHOD

METHOD PUBLIC SerializeWith
VAR_INPUT
	Serializer : I_Serializer;
END_VAR
Serializer.AddTod(activeData);
END_METHOD

PROPERTY PUBLIC Size : UDINT
GET
Size := SIZEOF(activeData);
END_GET
END_PROPERTY

METHOD TryDeserializeFrom : BOOL
VAR_INPUT
	Deserializer : I_Deserializer;
	Feedback : I_DeserializerFeedback;
END_VAR
TryDeserializeFrom := Deserializer.TryGetTod(activeData, Feedback);
END_METHOD

METHOD TryMakeReferenceTo : BOOL
VAR_INPUT
	Target : I_Datatype;
END_VAR
VAR
	pTargetData : POINTER TO TOD;
END_VAR
IF NOT (Target.IecType = IecType) THEN
	RETURN;
END_IF

pTargetData := Target.Address;
activeData REF= pTargetData^;
TryMakeReferenceTo := TRUE;
END_METHOD

PROPERTY PUBLIC Value : TOD
GET
Value := activeData;
END_GET
SET
activeData := Value;
END_SET
END_PROPERTY

END_FUNCTION_BLOCK

// Datatype/Primitive/_UDINT
{attribute 'linkalways'} 
{attribute 'no_explicit_call' := 'This FB is a CLASS and must be accessed using methods or properties'}
{attribute 'enable_dynamic_creation'}
FUNCTION_BLOCK _UDINT EXTENDS DatatypeBase
VAR
	localData : UDINT;
	activeData : REFERENCE TO UDINT REF= localData;
END_VAR

METHOD FB_init : BOOL
VAR_INPUT
	bInitRetains : BOOL; // if TRUE, the retain variables are initialized (warm start / cold start)
	bInCopyCode : BOOL;  // if TRUE, the instance afterwards gets moved into the copy code (online change)
	InitialValue : UDINT;
END_VAR
localData := InitialValue;
END_METHOD

PROPERTY PUBLIC Address : PVOID
GET
Address := ADR(activeData);
END_GET
END_PROPERTY

METHOD PUBLIC ClearReference
VAR_INPUT
END_VAR
activeData REF= localData;
END_METHOD

METHOD PUBLIC Clone : I_Datatype
VAR
    pClone : POINTER TO _UDINT;
END_VAR
pClone := __NEW(_UDINT(InitialValue := Value));
Clone := pClone^;
END_METHOD

PROPERTY PUBLIC IecType : T_MAXSTRING
GET
IecType := 'UDINT';
END_GET
END_PROPERTY

METHOD PUBLIC MakeReferenceTo
VAR_INPUT
	ReferenceTarget : REFERENCE TO UDINT;
END_VAR
activeData REF= ReferenceTarget;
END_METHOD

METHOD PUBLIC SerializeWith
VAR_INPUT
	Serializer : I_Serializer;
END_VAR
Serializer.AddUdint(activeData);
END_METHOD

PROPERTY PUBLIC Size : UDINT
GET
Size := SIZEOF(activeData);
END_GET
END_PROPERTY

METHOD TryDeserializeFrom : BOOL
VAR_INPUT
	Deserializer : I_Deserializer;
	Feedback : I_DeserializerFeedback;
END_VAR
TryDeserializeFrom := Deserializer.TryGetUdint(activeData, Feedback);
END_METHOD

METHOD TryMakeReferenceTo : BOOL
VAR_INPUT
	Target : I_Datatype;
END_VAR
VAR
	pTargetData : POINTER TO UDINT;
END_VAR
IF NOT (Target.IecType = IecType) THEN
	RETURN;
END_IF

pTargetData := Target.Address;
activeData REF= pTargetData^;
TryMakeReferenceTo := TRUE;
END_METHOD

PROPERTY PUBLIC Value : UDINT
GET
Value := activeData;
END_GET
SET
activeData := Value;
END_SET
END_PROPERTY

END_FUNCTION_BLOCK

// Datatype/Primitive/_UINT
{attribute 'linkalways'} 
{attribute 'no_explicit_call' := 'This FB is a CLASS and must be accessed using methods or properties'}
{attribute 'enable_dynamic_creation'}
FUNCTION_BLOCK _UINT EXTENDS DatatypeBase
VAR
	localData : UINT;
	activeData : REFERENCE TO UINT REF= localData;
END_VAR

METHOD FB_init : BOOL
VAR_INPUT
	bInitRetains : BOOL; // if TRUE, the retain variables are initialized (warm start / cold start)
	bInCopyCode : BOOL;  // if TRUE, the instance afterwards gets moved into the copy code (online change)
	InitialValue : UINT;
END_VAR
localData := InitialValue;
END_METHOD

PROPERTY PUBLIC Address : PVOID
GET
Address := ADR(activeData);
END_GET
END_PROPERTY

METHOD PUBLIC ClearReference
VAR_INPUT
END_VAR
activeData REF= localData;
END_METHOD

METHOD PUBLIC Clone : I_Datatype
VAR
    pClone : POINTER TO _UINT;
END_VAR
pClone := __NEW(_UINT(InitialValue := Value));
Clone := pClone^;
END_METHOD

PROPERTY PUBLIC IecType : T_MAXSTRING
GET
IecType := 'UINT';
END_GET
END_PROPERTY

METHOD PUBLIC MakeReferenceTo
VAR_INPUT
	ReferenceTarget : REFERENCE TO UINT;
END_VAR
activeData REF= ReferenceTarget;
END_METHOD

METHOD PUBLIC SerializeWith
VAR_INPUT
	Serializer : I_Serializer;
END_VAR
Serializer.AddUdint(activeData);
END_METHOD

PROPERTY PUBLIC Size : UDINT
GET
Size := SIZEOF(activeData);
END_GET
END_PROPERTY

METHOD TryDeserializeFrom : BOOL
VAR_INPUT
	Deserializer : I_Deserializer;
	Feedback : I_DeserializerFeedback;
END_VAR
TryDeserializeFrom := Deserializer.TryGetUint(activeData, Feedback);
END_METHOD

METHOD TryMakeReferenceTo : BOOL
VAR_INPUT
	Target : I_Datatype;
END_VAR
VAR
	pTargetData : POINTER TO UINT;
END_VAR
IF NOT (Target.IecType = IecType) THEN
	RETURN;
END_IF

pTargetData := Target.Address;
activeData REF= pTargetData^;
TryMakeReferenceTo := TRUE;
END_METHOD

PROPERTY PUBLIC Value : UINT
GET
Value := activeData;
END_GET
SET
activeData := Value;
END_SET
END_PROPERTY

END_FUNCTION_BLOCK

// Datatype/Primitive/_ULINT
{attribute 'linkalways'} 
{attribute 'no_explicit_call' := 'This FB is a CLASS and must be accessed using methods or properties'}
{attribute 'enable_dynamic_creation'}
FUNCTION_BLOCK _ULINT EXTENDS DatatypeBase
VAR
	localData : ULINT;
	activeData : REFERENCE TO ULINT REF= localData;
END_VAR

METHOD FB_init : BOOL
VAR_INPUT
	bInitRetains : BOOL; // if TRUE, the retain variables are initialized (warm start / cold start)
	bInCopyCode : BOOL;  // if TRUE, the instance afterwards gets moved into the copy code (online change)
	InitialValue : ULINT;
END_VAR
localData := InitialValue;
END_METHOD

PROPERTY PUBLIC Address : PVOID
GET
Address := ADR(activeData);
END_GET
END_PROPERTY

METHOD PUBLIC ClearReference
VAR_INPUT
END_VAR
activeData REF= localData;
END_METHOD

METHOD PUBLIC Clone : I_Datatype
VAR
    pClone : POINTER TO _ULINT;
END_VAR
pClone := __NEW(_ULINT(InitialValue := Value));
Clone := pClone^;
END_METHOD

PROPERTY PUBLIC IecType : T_MAXSTRING
GET
IecType := 'ULINT';
END_GET
END_PROPERTY

METHOD PUBLIC MakeReferenceTo
VAR_INPUT
	ReferenceTarget : REFERENCE TO ULINT;
END_VAR
activeData REF= ReferenceTarget;
END_METHOD

METHOD PUBLIC SerializeWith
VAR_INPUT
	Serializer : I_Serializer;
END_VAR
Serializer.AddUlint(activeData);
END_METHOD

PROPERTY PUBLIC Size : UDINT
GET
Size := SIZEOF(activeData);
END_GET
END_PROPERTY

METHOD TryDeserializeFrom : BOOL
VAR_INPUT
	Deserializer : I_Deserializer;
	Feedback : I_DeserializerFeedback;
END_VAR
TryDeserializeFrom := Deserializer.TryGetUlint(activeData, Feedback);
END_METHOD

METHOD TryMakeReferenceTo : BOOL
VAR_INPUT
	Target : I_Datatype;
END_VAR
VAR
	pTargetData : POINTER TO ULINT;
END_VAR
IF NOT (Target.IecType = IecType) THEN
	RETURN;
END_IF

pTargetData := Target.Address;
activeData REF= pTargetData^;
TryMakeReferenceTo := TRUE;
END_METHOD

PROPERTY PUBLIC Value : ULINT
GET
Value := activeData;
END_GET
SET
activeData := Value;
END_SET
END_PROPERTY

END_FUNCTION_BLOCK

// Datatype/Primitive/_USINT
{attribute 'linkalways'} 
{attribute 'no_explicit_call' := 'This FB is a CLASS and must be accessed using methods or properties'}
{attribute 'enable_dynamic_creation'}
FUNCTION_BLOCK _USINT EXTENDS DatatypeBase
VAR
	localData : USINT;
	activeData : REFERENCE TO USINT REF= localData;
END_VAR

METHOD FB_init : BOOL
VAR_INPUT
	bInitRetains : BOOL; // if TRUE, the retain variables are initialized (warm start / cold start)
	bInCopyCode : BOOL;  // if TRUE, the instance afterwards gets moved into the copy code (online change)
	InitialValue : USINT;
END_VAR
localData := InitialValue;
END_METHOD

PROPERTY PUBLIC Address : PVOID
GET
Address := ADR(activeData);
END_GET
END_PROPERTY

METHOD PUBLIC ClearReference
VAR_INPUT
END_VAR
activeData REF= localData;
END_METHOD

METHOD PUBLIC Clone : I_Datatype
VAR
    pClone : POINTER TO _USINT;
END_VAR
pClone := __NEW(_USINT(InitialValue := Value));
Clone := pClone^;
END_METHOD

PROPERTY PUBLIC IecType : T_MAXSTRING
GET
IecType := 'USINT';
END_GET
END_PROPERTY

METHOD PUBLIC MakeReferenceTo
VAR_INPUT
	ReferenceTarget : REFERENCE TO USINT;
END_VAR
activeData REF= ReferenceTarget;
END_METHOD

METHOD PUBLIC SerializeWith
VAR_INPUT
	Serializer : I_Serializer;
END_VAR
Serializer.AddUsint(activeData);
END_METHOD

PROPERTY PUBLIC Size : UDINT
GET
Size := SIZEOF(activeData);
END_GET
END_PROPERTY

METHOD TryDeserializeFrom : BOOL
VAR_INPUT
	Deserializer : I_Deserializer;
	Feedback : I_DeserializerFeedback;
END_VAR
TryDeserializeFrom := Deserializer.TryGetUsint(activeData, Feedback);
END_METHOD

METHOD TryMakeReferenceTo : BOOL
VAR_INPUT
	Target : I_Datatype;
END_VAR
VAR
	pTargetData : POINTER TO USINT;
END_VAR
IF NOT (Target.IecType = IecType) THEN
	RETURN;
END_IF

pTargetData := Target.Address;
activeData REF= pTargetData^;
TryMakeReferenceTo := TRUE;
END_METHOD

PROPERTY PUBLIC Value : USINT
GET
Value := activeData;
END_GET
SET
activeData := Value;
END_SET
END_PROPERTY

END_FUNCTION_BLOCK

// Datatype/Primitive/_WORD
{attribute 'linkalways'} 
{attribute 'no_explicit_call' := 'This FB is a CLASS and must be accessed using methods or properties'}
{attribute 'enable_dynamic_creation'}
FUNCTION_BLOCK _WORD EXTENDS DatatypeBase
VAR
	localData : WORD;
	activeData : REFERENCE TO WORD REF= localData;
END_VAR

METHOD FB_init : BOOL
VAR_INPUT
	bInitRetains : BOOL; // if TRUE, the retain variables are initialized (warm start / cold start)
	bInCopyCode : BOOL;  // if TRUE, the instance afterwards gets moved WORDo the copy code (online change)
	InitialValue : WORD;
END_VAR
localData := InitialValue;
END_METHOD

PROPERTY PUBLIC Address : PVOID
GET
Address := ADR(activeData);
END_GET
END_PROPERTY

METHOD PUBLIC ClearReference
VAR_INPUT
END_VAR
activeData REF= localData;
END_METHOD

METHOD PUBLIC Clone : I_Datatype
VAR
    pClone : POINTER TO _WORD;
END_VAR
pClone := __NEW(_WORD(InitialValue := Value));
Clone := pClone^;
END_METHOD

PROPERTY PUBLIC IecType : T_MAXSTRING
GET
IecType := 'WORD';
END_GET
END_PROPERTY

METHOD PUBLIC MakeReferenceTo
VAR_INPUT
	ReferenceTarget : REFERENCE TO WORD;
END_VAR
activeData REF= ReferenceTarget;
END_METHOD

METHOD PUBLIC SerializeWith
VAR_INPUT
	Serializer : I_Serializer;
END_VAR
Serializer.AddWord(activeData);
END_METHOD

PROPERTY PUBLIC Size : UDINT
GET
Size := SIZEOF(activeData);
END_GET
END_PROPERTY

METHOD TryDeserializeFrom : BOOL
VAR_INPUT
	Deserializer : I_Deserializer;
	Feedback : I_DeserializerFeedback;
END_VAR
TryDeserializeFrom := Deserializer.TryGetWord(activeData, Feedback);
END_METHOD

METHOD TryMakeReferenceTo : BOOL
VAR_INPUT
	Target : I_Datatype;
END_VAR
VAR
	pTargetData : POINTER TO WORD;
END_VAR
IF NOT (Target.IecType = IecType) THEN
	RETURN;
END_IF

pTargetData := Target.Address;
activeData REF= pTargetData^;
TryMakeReferenceTo := TRUE;
END_METHOD

PROPERTY PUBLIC Value : WORD
GET
Value := activeData;
END_GET
SET
activeData := Value;
END_SET
END_PROPERTY

END_FUNCTION_BLOCK

// Datatype/Structs/_TIMESTRUCT
{attribute 'linkalways'} 
{attribute 'no_explicit_call' := 'This FB is a CLASS and must be accessed using methods or properties'}
{attribute 'enable_dynamic_creation'}
FUNCTION_BLOCK _TIMESTRUCT EXTENDS StructuredDatatypeBase
VAR
	localData : TIMESTRUCT;
	activeData : REFERENCE TO TIMESTRUCT REF= localData;
	_wYear : _WORD(localData.wYear);
	_wMonth : _WORD(localData.wMonth);
	_wDayOfWeek : _WORD(localData.wDayOfWeek);
	_wDay : _WORD(localData.wDay);
	_wHour : _WORD(localData.wHour);
	_wMinute : _WORD(localData.wMinute);
	_wSecond : _WORD(localData.wSecond);
	_wMilliseconds : _WORD(localData.wMilliseconds);
END_VAR

METHOD FB_init : BOOL
VAR_INPUT
	bInitRetains : BOOL; // if TRUE, the retain variables are initialized (warm start / cold start)
	bInCopyCode : BOOL;  // if TRUE, the instance afterwards gets moved into the copy code (online change)
END_VAR
SetMemberReference();
AddMember('wYear',_wYear);
AddMember('wMonth',_wMonth);
AddMember('wDayOfWeek',_wDayOfWeek);
AddMember('wDay',_wDay);
AddMember('wHour',_wHour);
AddMember('wMinute',_wMinute);
AddMember('wSecond',_wSecond);
AddMember('wMilliseconds',_wMilliseconds);
END_METHOD

METHOD PROTECTED SetMemberReference
VAR_INPUT
END_VAR
_wYear.MakeReferenceTo(activeData.wYear);
_wMonth.MakeReferenceTo(activeData.wMonth);
_wDayOfWeek.MakeReferenceTo(activeData.wDayOfWeek);
_wDay.MakeReferenceTo(activeData.wDay);
_wHour.MakeReferenceTo(activeData.wHour);
_wMinute.MakeReferenceTo(activeData.wMinute);
_wSecond.MakeReferenceTo(activeData.wSecond);
_wMilliseconds.MakeReferenceTo(activeData.wMilliseconds);
END_METHOD

PROPERTY PUBLIC Address : PVOID
GET
Address := ADR(activeData);
END_GET
END_PROPERTY

METHOD PUBLIC ClearReference
VAR_INPUT
END_VAR
activeData REF= localData;
SetMemberReference();
END_METHOD

METHOD PUBLIC Clone : I_Datatype
VAR
    pClone : POINTER TO _TIMESTRUCT;
END_VAR
pClone := __NEW(_TIMESTRUCT());
pClone^.Value := Value;
Clone := pClone^;
END_METHOD

PROPERTY PUBLIC Identifier : T_MAXSTRING
GET
Identifier := 'TIMESTRUCT';
END_GET
END_PROPERTY

METHOD PUBLIC MakeReferenceTo
VAR_INPUT
	ReferenceTarget : REFERENCE TO TIMESTRUCT;
END_VAR
activeData REF= ReferenceTarget;
SetMemberReference();
END_METHOD

PROPERTY PUBLIC Size : UDINT
GET
Size := SIZEOF(activeData);
END_GET
END_PROPERTY

METHOD TryMakeReferenceTo : BOOL
VAR_INPUT
	Target : I_Datatype;
END_VAR
VAR
	pTargetData : POINTER TO TIMESTRUCT;
END_VAR
IF NOT (Target.IecType = IecType) THEN
	RETURN;
END_IF

pTargetData := Target.Address;
activeData REF= pTargetData^;
SetMemberReference();
TryMakeReferenceTo := TRUE;
END_METHOD

PROPERTY PUBLIC Value : TIMESTRUCT
GET
Value := activeData;
END_GET
SET
activeData := Value;
END_SET
END_PROPERTY

PROPERTY PUBLIC wDay : Reference to _WORD
GET
wDay REF= _wDay;
END_GET
END_PROPERTY

PROPERTY PUBLIC wDayOfWeek : Reference to _WORD
GET
wDayOfWeek REF= _wDayOfWeek;
END_GET
END_PROPERTY

PROPERTY PUBLIC wHour : Reference to _WORD
GET
wHour REF= _wHour;
END_GET
END_PROPERTY

PROPERTY PUBLIC wMilliseconds : Reference to _WORD
GET
wMilliseconds REF= _wMilliseconds;
END_GET
END_PROPERTY

PROPERTY PUBLIC wMinute : Reference to _WORD
GET
wMinute REF= _wMinute;
END_GET
END_PROPERTY

PROPERTY PUBLIC wMonth : Reference to _WORD
GET
wMonth REF= _wMonth;
END_GET
END_PROPERTY

PROPERTY PUBLIC wSecond : Reference to _WORD
GET
wSecond REF= _wSecond;
END_GET
END_PROPERTY

PROPERTY PUBLIC wYear : Reference to _WORD
GET
wYear REF= _wYear;
END_GET
END_PROPERTY

END_FUNCTION_BLOCK

// DatatypePacks/PlcBasicDatatypePack
{attribute 'linkalways'} 
{attribute 'no_explicit_call' := 'This FB is a CLASS and must be accessed using methods or properties'}
{attribute 'enable_dynamic_creation'}
FUNCTION_BLOCK PlcBasicDatatypePack IMPLEMENTS I_DatatypePack
VAR
	// alias
	_hresult : _HRESULT(0);
    _float : _FLOAT(0);
	
	// primitive
	_bool : _BOOL(FALSE);
	_byte : _BYTE(0);
	_dint : _DINT(0);
	_dt : _DT(DT#1970-1-1-0:0:0);
	_dword : _DWORD(0);
	_int : _INT(0);
	_lint : _LINT(0);
	_lreal : _LREAL(0);
	_lword : _LWORD(0);
	_real : _REAL(0);
	_sint : _SINT(0);
	_time_of_day : _TIME_OF_DAY(TOD#0:0:0);
	_tod : _TOD(TOD#0:0:0);
	_udint : _UDINT(0);
	_uint : _UINT(0);
	_ulint : _ULINT(0);
	_usint : _USINT(0);
	_word : _WORD(0);
	
	// structures
	_timestruct : _TIMESTRUCT();
	
END_VAR

METHOD RegisterWith
VAR_INPUT
	Datatypes : I_Datatypes;
END_VAR
// alias
Datatypes.RegisterDatatype(_hresult);
Datatypes.RegisterDatatype(_float);

// primitive
Datatypes.RegisterDatatype(_bool);
Datatypes.RegisterDatatype(_byte);
Datatypes.RegisterDatatype(_dint);
Datatypes.RegisterDatatype(_dt);
Datatypes.RegisterDatatype(_dword);
Datatypes.RegisterDatatype(_int);
Datatypes.RegisterDatatype(_lint);
Datatypes.RegisterDatatype(_lreal);
Datatypes.RegisterDatatype(_lword);
Datatypes.RegisterDatatype(_real);
Datatypes.RegisterDatatype(_sint);
Datatypes.RegisterDatatype(_time_of_day);
Datatypes.RegisterDatatype(_tod);
Datatypes.RegisterDatatype(_udint);
Datatypes.RegisterDatatype(_uint);
Datatypes.RegisterDatatype(_ulint);
Datatypes.RegisterDatatype(_usint);
Datatypes.RegisterDatatype(_word);

// structures
Datatypes.RegisterDatatype(_timestruct);
END_METHOD

END_FUNCTION_BLOCK

// Interfaces/I_DatatypePack
INTERFACE I_DatatypePack

METHOD RegisterWith
VAR_INPUT
	Datatypes : I_Datatypes;
END_VAR
END_METHOD

END_INTERFACE

// Datatypes/Datatypes
{attribute 'linkalways'} 
{attribute 'no_explicit_call' := 'This FB is a CLASS and must be accessed using methods or properties'}
{attribute 'enable_dynamic_creation'}
FUNCTION_BLOCK Datatypes IMPLEMENTS I_Datatypes
VAR
	primitives : Dictionary;
	structures : Dictionary;
	alias : Dictionary;
END_VAR

METHOD PRIVATE SerializeAliasTypeWith
VAR_INPUT
	Serializer : I_Serializer;
END_VAR
VAR
	enumerator : I_ForwardEnumerator;
	datatype : I_AliasDatatype;
END_VAR
enumerator := alias.GetEnumerator();

WHILE enumerator.MoveNext() DO
	IF enumerator.TryGet(datatype) THEN
		datatype.SerializeTypeWith(Serializer);
	END_IF
END_WHILE

enumerator.Dispose();
END_METHOD

METHOD PRIVATE SerializePrimitiveTypeWith
VAR_INPUT
	Serializer : I_Serializer;
END_VAR
VAR
	enumerator : I_ForwardEnumerator;
	datatype : I_Datatype;
END_VAR
enumerator := primitives.GetEnumerator();

WHILE enumerator.MoveNext() DO
	IF enumerator.TryGet(datatype) THEN
		datatype.SerializeTypeWith(Serializer);
	END_IF
END_WHILE

enumerator.Dispose();
END_METHOD

METHOD PRIVATE SerializeStructuresTypeWith
VAR_INPUT
	Serializer : I_Serializer;
END_VAR
VAR
	enumerator : I_ForwardEnumerator;
	datatype : I_StructuredDatatype;
END_VAR
enumerator := structures.GetEnumerator();

WHILE enumerator.MoveNext() DO
	IF enumerator.TryGet(datatype) THEN
		datatype.SerializeTypeWith(Serializer);
	END_IF
END_WHILE

enumerator.Dispose();
END_METHOD

METHOD PUBLIC GetAliasByIdentifier : BOOL
VAR_INPUT
	Identifier : T_MAXSTRING;
	Destination : REFERENCE TO I_AliasDatatype;
END_VAR
GetAliasByIdentifier := alias.TryGetValue(Identifier, Destination);
END_METHOD

METHOD PUBLIC GetPrimitiveByIecType : BOOL
VAR_INPUT
	Identifier : T_MAXSTRING;
	Destination : REFERENCE TO I_AliasDatatype;
END_VAR
GetPrimitiveByIecType := primitives.TryGetValue(Identifier, Destination);
END_METHOD

METHOD PUBLIC GetStructureByIdentifier : BOOL
VAR_INPUT
	Identifier : T_MAXSTRING;
	Destination : REFERENCE TO I_StructuredDatatype;
END_VAR
GetStructureByIdentifier := structures.TryGetValue(Identifier, Destination);
END_METHOD

METHOD RegisterDatatype
VAR_INPUT
	Datatype : I_Datatype;
END_VAR
VAR
	datatypeAsStructure : I_StructuredDatatype;
	datatypeAsAlias : I_AliasDatatype;
END_VAR
IF Datatype.TryResolveAsStructuredType(datatypeAsStructure) THEN
	structures.AddOrUpdate(datatypeAsStructure.Identifier, datatypeAsStructure);
	RETURN;
END_IF

IF Datatype.TryResolveAsAliasType(datatypeAsAlias) THEN
	alias.AddOrUpdate(datatypeAsAlias.Identifier, datatypeAsAlias);
	RETURN;
END_IF

// add enumeration

// add arrays

primitives.AddOrUpdate(Datatype.IecType, Datatype);
END_METHOD

METHOD PUBLIC SerializeTypeWith
VAR_INPUT
	Serializer : I_Serializer;
END_VAR
Serializer.StartObject();
Serializer.AddKey('datatypes');
Serializer.StartArray();
SerializePrimitiveTypeWith(Serializer);
SerializeStructuresTypeWith(Serializer);
SerializeAliasTypeWith(Serializer);
Serializer.EndArray();
Serializer.EndObject();
END_METHOD

END_FUNCTION_BLOCK

// Interfaces/I_Datatypes
INTERFACE I_Datatypes

METHOD PUBLIC GetAliasByIdentifier : BOOL
VAR_INPUT
	Identifier : T_MAXSTRING;
	Destination : REFERENCE TO I_AliasDatatype;
END_VAR
END_METHOD

METHOD PUBLIC GetPrimitiveByIecType : BOOL
VAR_INPUT
	Identifier : T_MAXSTRING;
	Destination : REFERENCE TO I_AliasDatatype;
END_VAR
END_METHOD

METHOD PUBLIC GetStructureByIdentifier : BOOL
VAR_INPUT
	Identifier : T_MAXSTRING;
	Destination : REFERENCE TO I_StructuredDatatype;
END_VAR
END_METHOD

METHOD RegisterDatatype
VAR_INPUT
	Datatype : I_Datatype;
END_VAR
END_METHOD

METHOD PUBLIC SerializeTypeWith
VAR_INPUT
	Serializer : I_Serializer;
END_VAR
END_METHOD

END_INTERFACE
